(*
SPDX-FileCopyrightText: © 2026 Oleksandr Tiutyk <trofimich@gmail.com>
SPDX-License-Identifier: MIT
License: https://opensource.org/license/mit
*)

INTERFACE IJsonExtender

METHOD ExtendAtFinish
VAR_IN_OUT CONSTANT
	jsonSaxWriter : Tc3_JsonXml.FB_JsonSaxWriter;	
END_VAR
END_METHOD

METHOD ExtendAtStart
VAR_IN_OUT CONSTANT
	jsonSaxWriter : Tc3_JsonXml.FB_JsonSaxWriter;	
END_VAR
END_METHOD

END_INTERFACE

(* stored: Version 1.1.0.1
   Itf IJsonExtender: Id {4855e1bf-29d3-434d-ad18-57cfe564a05a}
   Method ExtendAtFinish: Id {3bd84534-1712-40b5-9503-1fc6ee164105}
   Method ExtendAtStart: Id {9509cef5-06c5-4632-a66c-dbe1c085047e} *)
